// TwinCAT 3 PLC project TcDeviceBase
// Title: TcDeviceBase
// Company: TcNexa
// Author: ATI Software Engineering
// ProjectVersion: 2.0.0
// ProgramVersion: 3.1.4026.19
// libraries:
//   Tc2_Standard, * (Beckhoff Automation GmbH)
//   Tc2_System, * (Beckhoff Automation GmbH)
//   Tc3_IotBase, * (Beckhoff Automation GmbH)
//   Tc3_Module, * (Beckhoff Automation GmbH)
//   TcNexaHmi, * (TcNexa)
//   TcProcess, * (TcNexa)
//   TcUtilities, * (TcNexa)
// project tree:
//   Base/DUTs/ ST_MethodState.TcDUT
//   Base/POUs/ FB_DeviceBase.TcPOU (not stored), FB_DeviceNexaHmi.TcPOU (not stored)
//   Components/ FB_DeviceButtonNexaHmi.TcPOU (not stored)
//   / PlcTask.TcTTO
//   Tests/ PRG_TEST.TcPOU (not stored)
//   Version/ Global_Version.TcGVL
// real-time tasks:
//   TASK PlcTask: cycle T#10ms, priority 20, ADS port 350

CONFIGURATION TcDeviceBase
    RESOURCE PLC ON TwinCAT3
        TASK PlcTask(INTERVAL := T#10ms, PRIORITY := 20);
        PROGRAM PRG_TEST WITH PlcTask : PRG_TEST;
    END_RESOURCE
END_CONFIGURATION

// ---- Base/DUTs/ST_MethodState.TcDUT
TYPE ST_MethodState :
STRUCT
	init		: BOOL;
	execute		: BOOL;
	timeout		: BOOL;
END_STRUCT
END_TYPE

// ---- Version/Global_Version.TcGVL
{attribute 'TcGenerated'}
{attribute 'no-analysis'}
{attribute 'linkalways'}
// This function has been automatically generated from the project information.
VAR_GLOBAL CONSTANT
	{attribute 'const_non_replaced'}
	stLibVersion_TcDeviceBase : ST_LibVersion := (iMajor := 2, iMinor := 0, iBuild := 0, iRevision := 0, nFlags := 0, sVersion := '2.0.0');
END_VAR
